// SIMATIC S7-200 project (STEP 7-Micro/WIN), CPU 221 REL 01.10

SYMBOL_TABLE USER1
PBR              I0.0
PBL              I0.1
DC0              Q0.0
DC1              Q0.1
DC2              Q0.2
DC3              Q0.3
DC4              Q0.4
DC5              Q0.5
DC6              Q0.6
DC7              Q0.7
END_SYMBOL_TABLE

ORGANIZATION_BLOCK MAIN:OB1
TITLE=
BEGIN
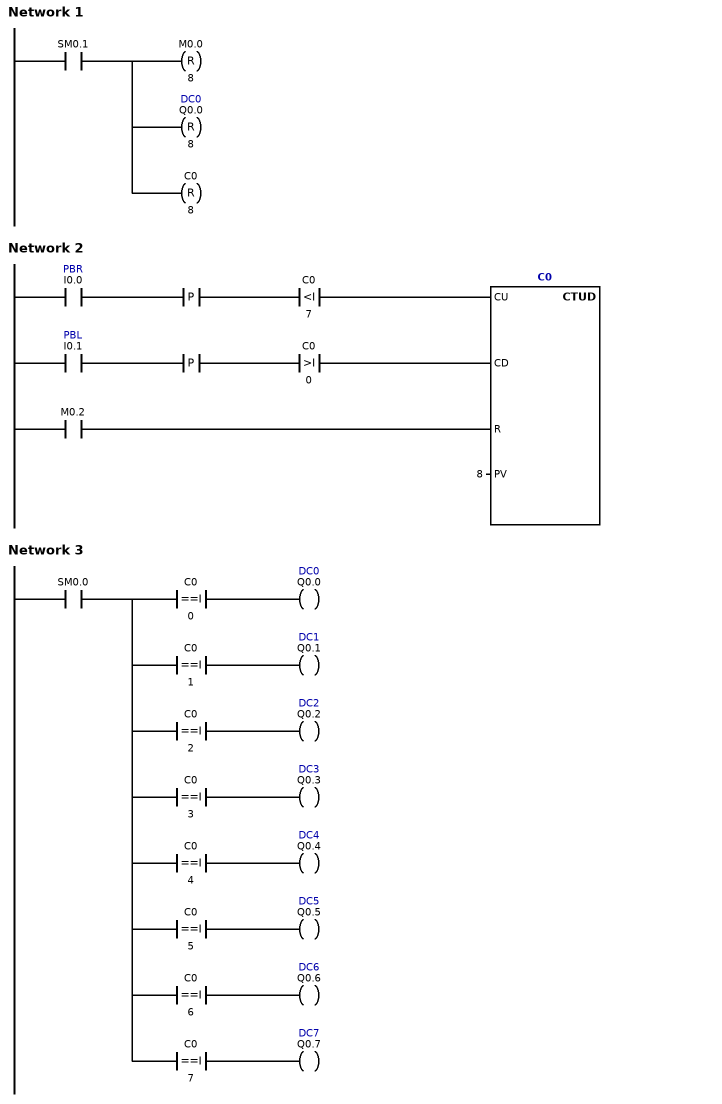
Network 1
LD     SM0.1
R      M0.0, 8
R      DC0:Q0.0, 8
R      C0, 8
Network 2
LD     PBR:I0.0
EU
AW<    C0, 7
LD     PBL:I0.1
EU
AW>    C0, 0
LD     M0.2
CTUD   C0, 8
Network 3
LD     SM0.0
LPS
AW=    C0, 0
=      DC0:Q0.0
LRD
AW=    C0, 1
=      DC1:Q0.1
LRD
AW=    C0, 2
=      DC2:Q0.2
LRD
AW=    C0, 3
=      DC3:Q0.3
LRD
AW=    C0, 4
=      DC4:Q0.4
LRD
AW=    C0, 5
=      DC5:Q0.5
LRD
AW=    C0, 6
=      DC6:Q0.6
LPP
AW=    C0, 7
=      DC7:Q0.7
END_ORGANIZATION_BLOCK
